{attribute 'GeneratedUsingTerminal: AT2050-0501-0020'}
{attribute addProperty BoxType "AT2050-0501-0020"}
{attribute addProperty Id "A_0087_AT2050_5501_0016_AT2050_5501AT2050_33A3DF1B80"}
{attribute addProperty CRC "2851410171"}
{attribute addProperty Size "80"}
TYPE A_0057_AT2050_0501_0020_A9F510FB EXTENDS AT2050_A7FEA1CF :
STRUCT
	{attribute addProperty Name "A_0087_AT2050_5501_0016_AT2050_5501"}
	{attribute addProperty PreviousPort "A_0057(AT2050-0501-0020) : B"}
	A_0087_AT2050_5501_0016_AT2050_5501 : AT2050_33A3DF1B;
END_STRUCT
END_TYPE

(* stored: Version 1.2.0.0, ProductVersion 3.1.4024.9
   DUT A_0057_AT2050_0501_0020_A9F510FB: Id {b962f8aa-ccaa-4b0b-bc08-9982d21a6074} *)
